FUNCTION_BLOCK FB_Machine
VAR_INPUT
END_VAR
VAR_OUTPUT

END_VAR
VAR
	Tower : FB_Tower;
	//fManualLowSpeed		: LREAL;
	//fManualHighSpeed	: LREAL;	
	
END_VAR

Tower();

(*
MCJog( Axis := 	stAxis, Velocity := fManualVelocity, Mode := MC_JOGMODE_CONTINOUS );				
McPower(Axis := stAxis);
McReset(Axis := stAxis); 
ActUpdateAxisData();
ActUpdateManVelocity();


CASE GVL.eMachineState OF
	

	// The machine starts up in Error state
	E_MachineState.Error:	
	
	// Changes statet to Ready state
	IF startButton THEN
		readyLamp := TRUE;
		SetState( E_MachineState.Ready );
	END_IF
	
	
	
	E_MachineState.Ready:
	McReset.Execute := TRUE;
		IF McReset.Done THEN 
			McReset.Execute := FALSE; 
		END_IF 	
	
		IF (ActualPos < lowerLimit OR ActualPos > upperLimit) AND enableButton THEN
			 
			IF ActualPos > upperLimit AND enableButton THEN
				McPower.Enable 			:= TRUE;
				McPower.Enable_Negative := TRUE;
				SetState( E_MachineState.Running );
			END_IF
			
			IF ActualPos < lowerLimit AND enableButton THEN 
				McPower.Enable 			:= TRUE;
				McPower.Enable_Positive := TRUE;
				SetState( E_MachineState.Running );
			END_IF
		END_IF
		
 		// Enables the axis for movement
		IF enableButton AND ActualPos > lowerLimit AND ActualPos < upperLimit  THEN
			McPower.Enable 			:= TRUE;
			McPower.Enable_Positive := TRUE; 
			McPower.Enable_Negative := TRUE;		
			SetState( E_MachineState.Running );
		END_IF
		
		// Disables the axis for movement
		IF stopButton THEN
			McPower.Enable 			:= FALSE;
			McPower.Enable_Positive := FALSE; 
			McPower.Enable_Negative := FALSE;
			enableButton 			:= FALSE;
			MCJog.JogForward 		:= FALSE; 
			MCJog.JogBackwards 		:= FALSE;
		END_IF
			
			
	E_MachineState.Running: 	
		
		// forward and backward movement logic
		IF forwardButton OR backwardButton THEN
			IF (ActualPos > lowerLimit AND ActualPos < upperLimit) THEN 
				McPower.Enable_Positive := TRUE; 
				McPower.Enable_Negative := TRUE;
			END_IF 
			IF forwardButton THEN 
				MCJog.JogForward 	:= TRUE;
				MCJog.JogBackwards 	:= FALSE;
			END_IF 
			
			IF backwardButton THEN
				MCJog.JogBackwards 	:= TRUE; 
				MCJog.JogForward 	:= FALSE;
			END_IF 
		ELSE 
			MCJog.JogBackwards 	:= FALSE;
			MCJog.JogForward 	:= FALSE;
		END_IF
		
		// Disables the axis for movement
		IF stopButton THEN
			McPower.Enable 			:= FALSE;
			McPower.Enable_Positive := FALSE; 
			McPower.Enable_Negative := FALSE;
			enableButton 			:= FALSE;
			MCJog.JogForward 		:= FALSE; 
			MCJog.JogBackwards 		:= FALSE;
	
			SetState( E_MachineState.Ready );
		END_IF  
		
		IF (ActualPos < lowerLimit OR ActualPos > upperLimit) AND McPower.Enable_Positive AND McPower.Enable_Negative THEN 
			McPower.Enable 			:= FALSE;
			McPower.Enable_Positive := FALSE; 
			McPower.Enable_Negative := FALSE;
			enableButton 			:= FALSE;
			MCJog.JogForward 		:= FALSE; 
			MCJog.JogBackwards 		:= FALSE;
	
			SetState( E_MachineState.Error );
		END_IF
		

END_CASE

*)

END_FUNCTION_BLOCK

(* stored: Version 1.1.0.1, ProductVersion 3.1.4024.9
   POU FB_Machine: Id {7ef33cb4-4633-4fdb-af8e-925e40a544a1}, SpecialFunc None *)
